// Mitsubishi GX Works2 project: 시퀀스 회로 예제 (타이머)   PLC: Q03UDV

PROGRAM MAIN
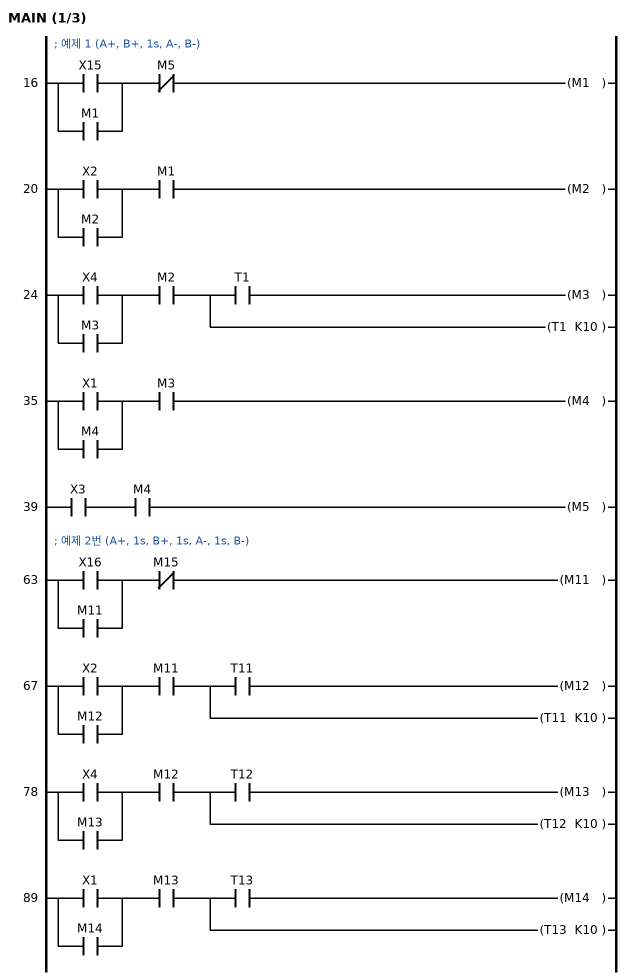
; 예제 1 (A+, B+, 1s, A-, B-)
16    LD      X15
      OR      M1
      ANI     M5
      OUT     M1
20    LD      X2
      OR      M2
      AND     M1
      OUT     M2
24    LD      X4
      OR      M3
      AND     M2
      MPS
      AND     T1
      OUT     M3
      MPP
      OUT     T1 K10
35    LD      X1
      OR      M4
      AND     M3
      OUT     M4
39    LD      X3
      AND     M4
      OUT     M5
; 예제 2번 (A+, 1s, B+, 1s, A-, 1s, B-)
63    LD      X16
      OR      M11
      ANI     M15
      OUT     M11
67    LD      X2
      OR      M12
      AND     M11
      MPS
      AND     T11
      OUT     M12
      MPP
      OUT     T11 K10
78    LD      X4
      OR      M13
      AND     M12
      MPS
      AND     T12
      OUT     M13
      MPP
      OUT     T12 K10
89    LD      X1
      OR      M14
      AND     M13
      MPS
      AND     T13
      OUT     M14
      MPP
      OUT     T13 K10
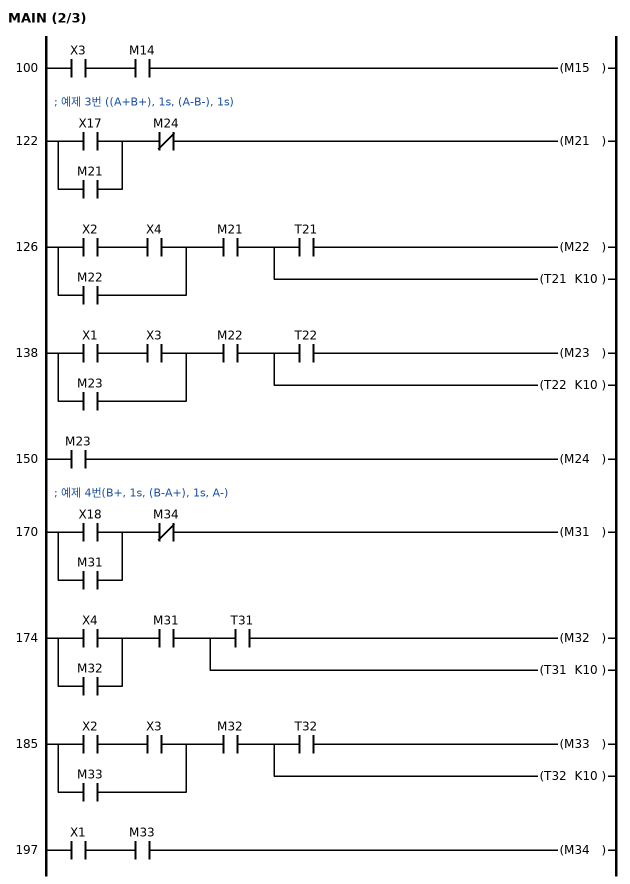
100   LD      X3
      AND     M14
      OUT     M15
; 예제 3번 ((A+B+), 1s, (A-B-), 1s)
122   LD      X17
      OR      M21
      ANI     M24
      OUT     M21
126   LD      X2
      AND     X4
      OR      M22
      AND     M21
      MPS
      AND     T21
      OUT     M22
      MPP
      OUT     T21 K10
138   LD      X1
      AND     X3
      OR      M23
      AND     M22
      MPS
      AND     T22
      OUT     M23
      MPP
      OUT     T22 K10
150   LD      M23
      OUT     M24
; 예제 4번(B+, 1s, (B-A+), 1s, A-)
170   LD      X18
      OR      M31
      ANI     M34
      OUT     M31
174   LD      X4
      OR      M32
      AND     M31
      MPS
      AND     T31
      OUT     M32
      MPP
      OUT     T31 K10
185   LD      X2
      AND     X3
      OR      M33
      AND     M32
      MPS
      AND     T32
      OUT     M33
      MPP
      OUT     T32 K10
197   LD      X1
      AND     M33
      OUT     M34
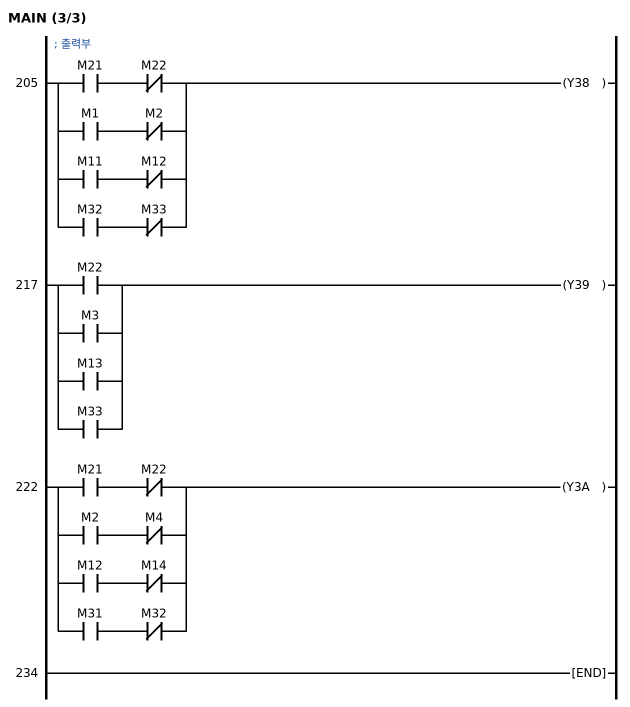
; 출력부
205   LD      M21
      ANI     M22
      LD      M1
      ANI     M2
      ORB
      LD      M11
      ANI     M12
      ORB
      LD      M32
      ANI     M33
      ORB
      OUT     Y38
217   LD      M22
      OR      M3
      OR      M13
      OR      M33
      OUT     Y39
222   LD      M21
      ANI     M22
      LD      M2
      ANI     M4
      ORB
      LD      M12
      ANI     M14
      ORB
      LD      M31
      ANI     M32
      ORB
      OUT     Y3A
234   END
END_PROGRAM
